PROGRAM MAIN_XYZ
VAR
	
END_VAR

//main program for gcode
	//POU_NCI();

//JSON
	decCOM();
	readJSONfile();
	decFile();

//AT Commands
	commandDecoder();
	commandExecute();

//Error
	ERROR();

MAIN_MQTT();

END_PROGRAM

(* stored: Version 1.1.0.1, ProductVersion 3.1.4024.2
   POU MAIN_XYZ: Id {f3e90440-582f-45a4-ac51-5f2449296ba8}, SpecialFunc None *)
